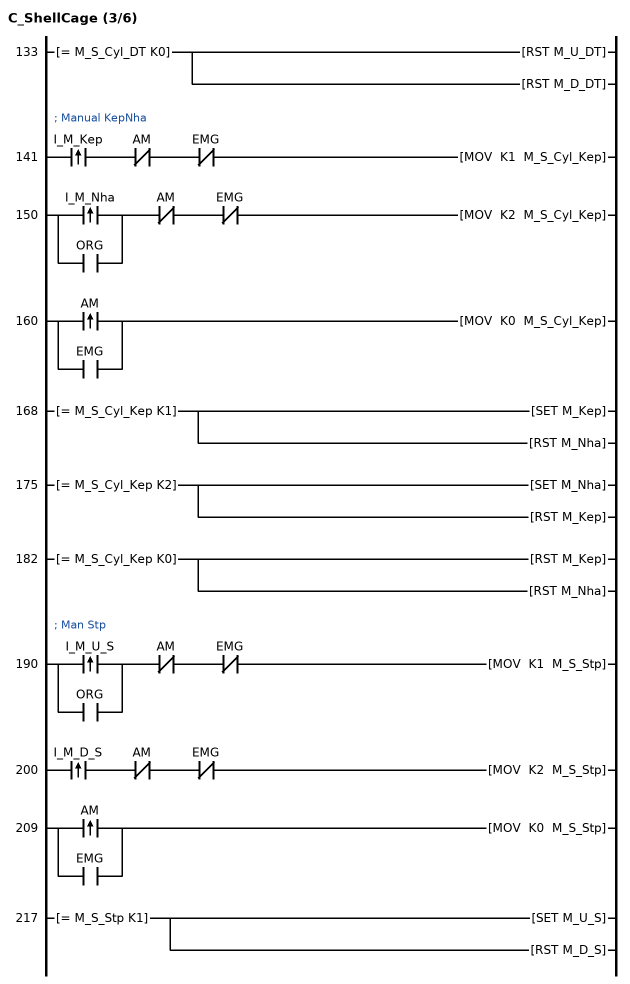
[picture p48: ladder of C_ShellCage, rungs at steps 133 to 217]
133   LD=     M_S_Cyl_DT K0
      RST     M_U_DT
      RST     M_D_DT
; Manual KepNha
141   LDP     I_M_Kep
      ANI     AM
      ANI     EMG
      MOV     K1 M_S_Cyl_Kep
150   LDP     I_M_Nha
      OR      ORG
      ANI     AM
      ANI     EMG
      MOV     K2 M_S_Cyl_Kep
160   LDP     AM
      OR      EMG
      MOV     K0 M_S_Cyl_Kep
168   LD=     M_S_Cyl_Kep K1
      SET     M_Kep
      RST     M_Nha
175   LD=     M_S_Cyl_Kep K2
      SET     M_Nha
      RST     M_Kep
182   LD=     M_S_Cyl_Kep K0
      RST     M_Kep
      RST     M_Nha
; Man Stp
190   LDP     I_M_U_S
      OR      ORG
      ANI     AM
      ANI     EMG
      MOV     K1 M_S_Stp
200   LDP     I_M_D_S
      ANI     AM
      ANI     EMG
      MOV     K2 M_S_Stp
209   LDP     AM
      OR      EMG
      MOV     K0 M_S_Stp
217   LD=     M_S_Stp K1
      SET     M_U_S
      RST     M_D_S
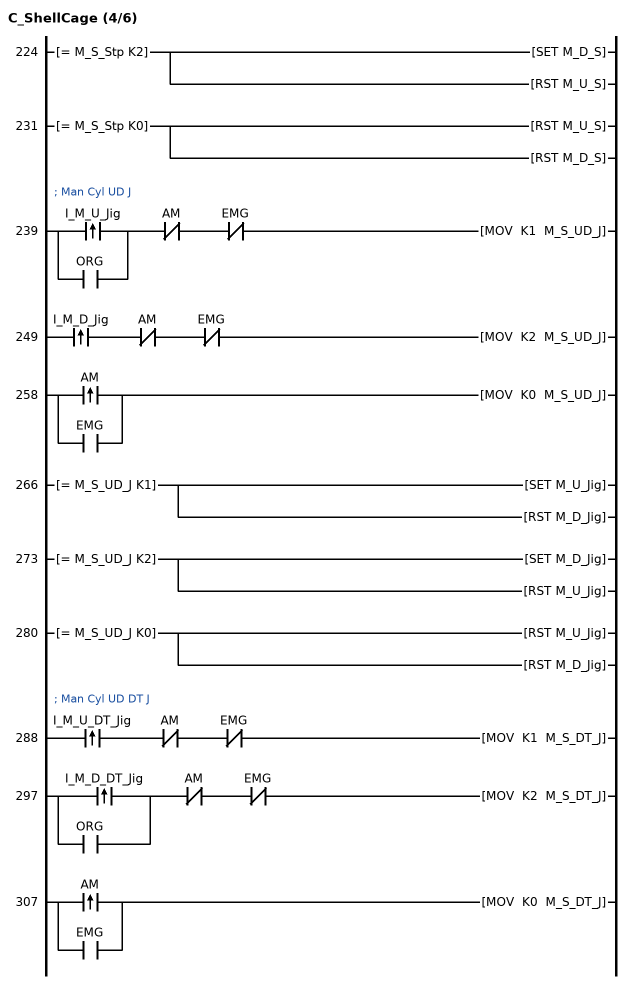
224   LD=     M_S_Stp K2
      SET     M_D_S
      RST     M_U_S
231   LD=     M_S_Stp K0
      RST     M_U_S
      RST     M_D_S
; Man Cyl UD J
239   LDP     I_M_U_Jig
      OR      ORG
      ANI     AM
      ANI     EMG
      MOV     K1 M_S_UD_J
249   LDP     I_M_D_Jig
      ANI     AM
      ANI     EMG
      MOV     K2 M_S_UD_J
258   LDP     AM
      OR      EMG
      MOV     K0 M_S_UD_J
266   LD=     M_S_UD_J K1
      SET     M_U_Jig
      RST     M_D_Jig
273   LD=     M_S_UD_J K2
      SET     M_D_Jig
      RST     M_U_Jig
280   LD=     M_S_UD_J K0
      RST     M_U_Jig
      RST     M_D_Jig
; Man Cyl UD DT J
288   LDP     I_M_U_DT_Jig
      ANI     AM
      ANI     EMG
      MOV     K1 M_S_DT_J
297   LDP     I_M_D_DT_Jig
      OR      ORG
      ANI     AM
      ANI     EMG
      MOV     K2 M_S_DT_J
307   LDP     AM
      OR      EMG
      MOV     K0 M_S_DT_J
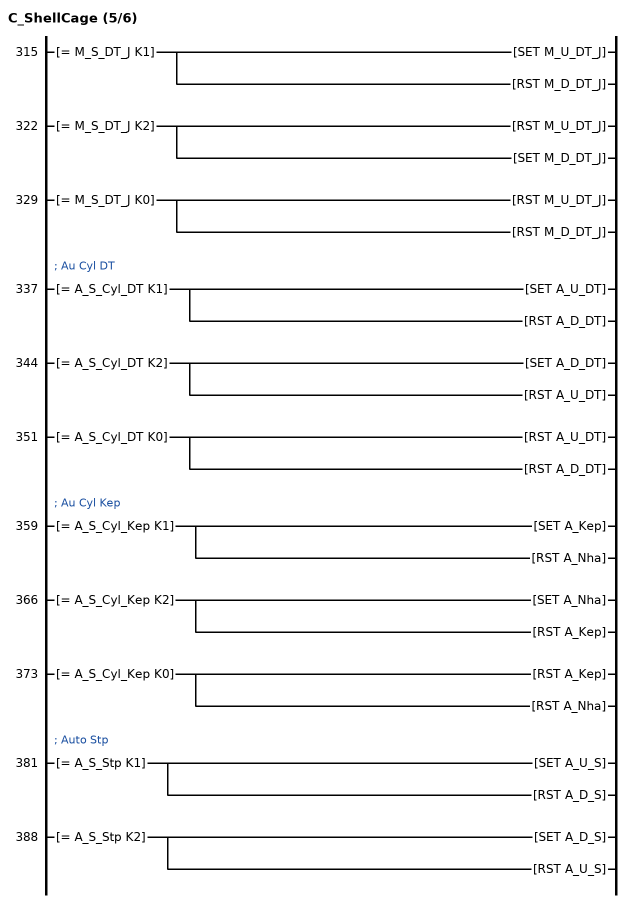
315   LD=     M_S_DT_J K1
      SET     M_U_DT_J
      RST     M_D_DT_J
322   LD=     M_S_DT_J K2
      RST     M_U_DT_J
      SET     M_D_DT_J
329   LD=     M_S_DT_J K0
      RST     M_U_DT_J
      RST     M_D_DT_J
; Au Cyl DT
337   LD=     A_S_Cyl_DT K1
      SET     A_U_DT
      RST     A_D_DT
344   LD=     A_S_Cyl_DT K2
      SET     A_D_DT
      RST     A_U_DT
351   LD=     A_S_Cyl_DT K0
      RST     A_U_DT
      RST     A_D_DT
; Au Cyl Kep
359   LD=     A_S_Cyl_Kep K1
      SET     A_Kep
      RST     A_Nha
366   LD=     A_S_Cyl_Kep K2
      SET     A_Nha
      RST     A_Kep
373   LD=     A_S_Cyl_Kep K0
      RST     A_Kep
      RST     A_Nha
; Auto Stp
381   LD=     A_S_Stp K1
      SET     A_U_S
      RST     A_D_S
388   LD=     A_S_Stp K2
      SET     A_D_S
      RST     A_U_S
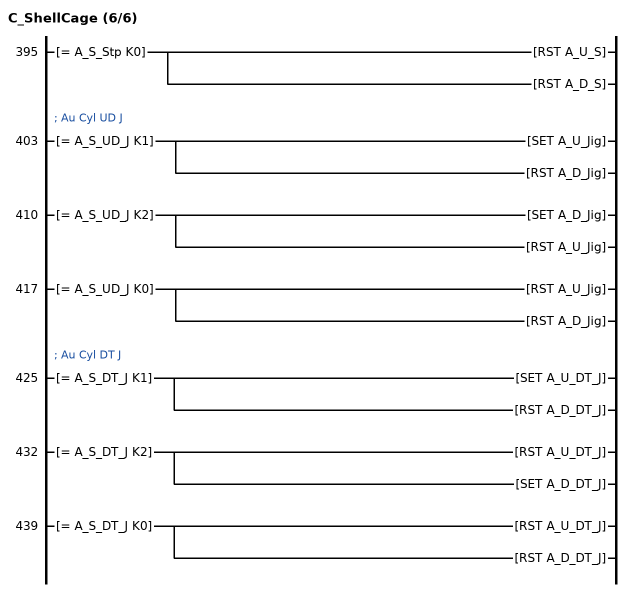
395   LD=     A_S_Stp K0
      RST     A_U_S
      RST     A_D_S
; Au Cyl UD J
403   LD=     A_S_UD_J K1
      SET     A_U_Jig
      RST     A_D_Jig
410   LD=     A_S_UD_J K2
      SET     A_D_Jig
      RST     A_U_Jig
417   LD=     A_S_UD_J K0
      RST     A_U_Jig
      RST     A_D_Jig
; Au Cyl DT J
425   LD=     A_S_DT_J K1
      SET     A_U_DT_J
      RST     A_D_DT_J
432   LD=     A_S_DT_J K2
      RST     A_U_DT_J
      SET     A_D_DT_J
439   LD=     A_S_DT_J K0
      RST     A_U_DT_J
      RST     A_D_DT_J
END_FUNCTION_BLOCK

PROGRAM Position
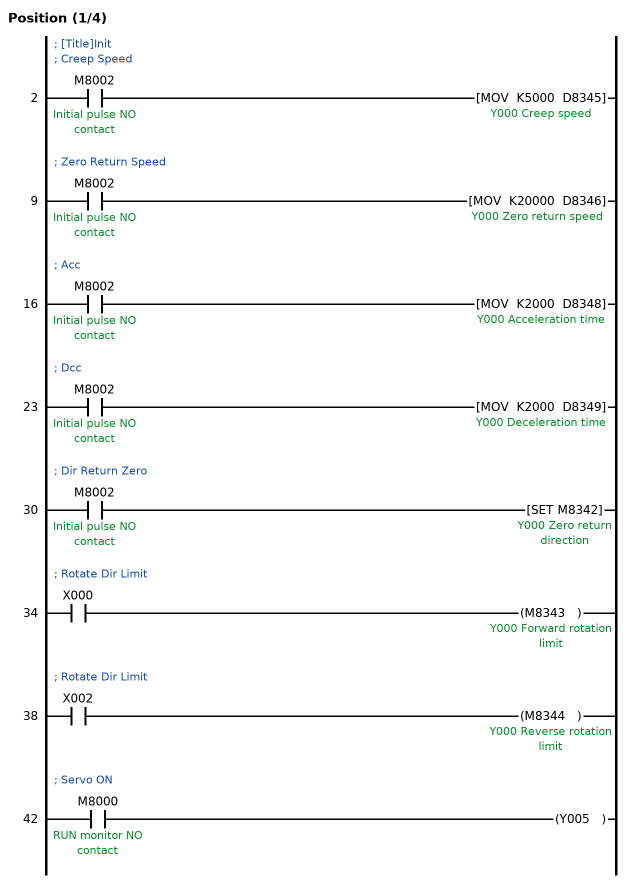
; [Title]Init
; Creep Speed
2     LD      M8002  ; Initial pulse NO contact
      MOV     K5000 D8345  ; Y000 Creep speed
; Zero Return Speed
9     LD      M8002  ; Initial pulse NO contact
      MOV     K20000 D8346  ; Y000 Zero return speed
; Acc
16    LD      M8002  ; Initial pulse NO contact
      MOV     K2000 D8348  ; Y000 Acceleration time
; Dcc
23    LD      M8002  ; Initial pulse NO contact
      MOV     K2000 D8349  ; Y000 Deceleration time
; Dir Return Zero
30    LD      M8002  ; Initial pulse NO contact
      SET     M8342  ; Y000 Zero return direction
; Rotate Dir Limit
34    LD      X000
      OUT     M8343  ; Y000 Forward rotation limit
; Rotate Dir Limit
38    LD      X002
      OUT     M8344  ; Y000 Reverse rotation limit
; Servo ON
42    LD      M8000  ; RUN monitor NO contact
      OUT     Y005
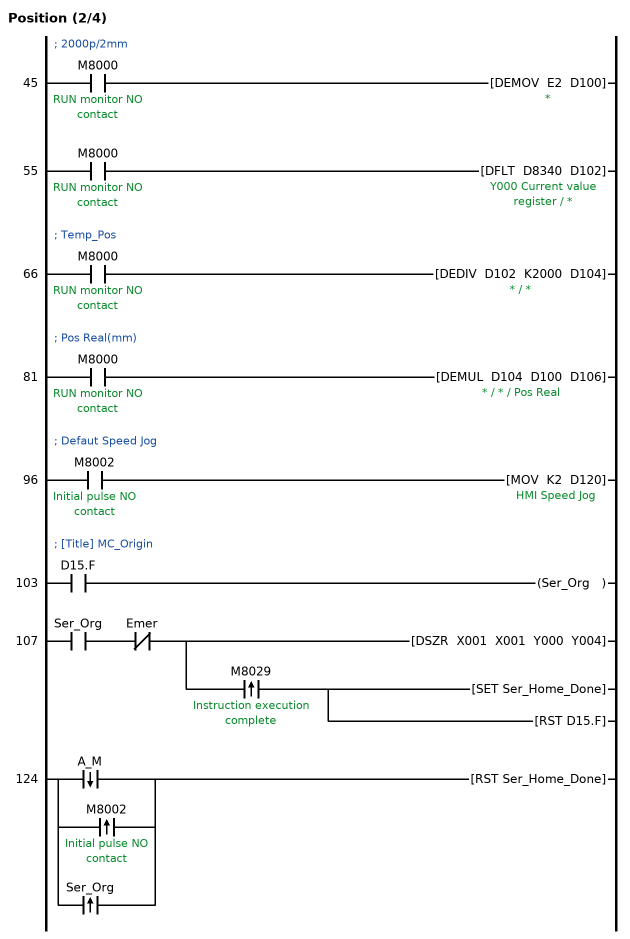
; 2000p/2mm
45    LD      M8000  ; RUN monitor NO contact
      DEMOV   E2 D100  ; *
55    LD      M8000  ; RUN monitor NO contact
      DFLT    D8340 D102  ; Y000 Current value register / *
; Temp_Pos
66    LD      M8000  ; RUN monitor NO contact
      DEDIV   D102 K2000 D104  ; *
; Pos Real(mm)
81    LD      M8000  ; RUN monitor NO contact
      DEMUL   D104 D100 D106  ; Pos Real
; Defaut Speed Jog
96    LD      M8002  ; Initial pulse NO contact
      MOV     K2 D120  ; HMI Speed Jog
; [Title] MC_Origin
103   LD      D15.F
      OUT     Ser_Org
107   LD      Ser_Org
      ANI     Emer
      DSZR    X001 X001 Y000 Y004
      ANDP    M8029  ; Instruction execution complete
      SET     Ser_Home_Done
      RST     D15.F
124   LDF     A_M
      ORP     M8002  ; Initial pulse NO contact
      ORP     Ser_Org
      RST     Ser_Home_Done
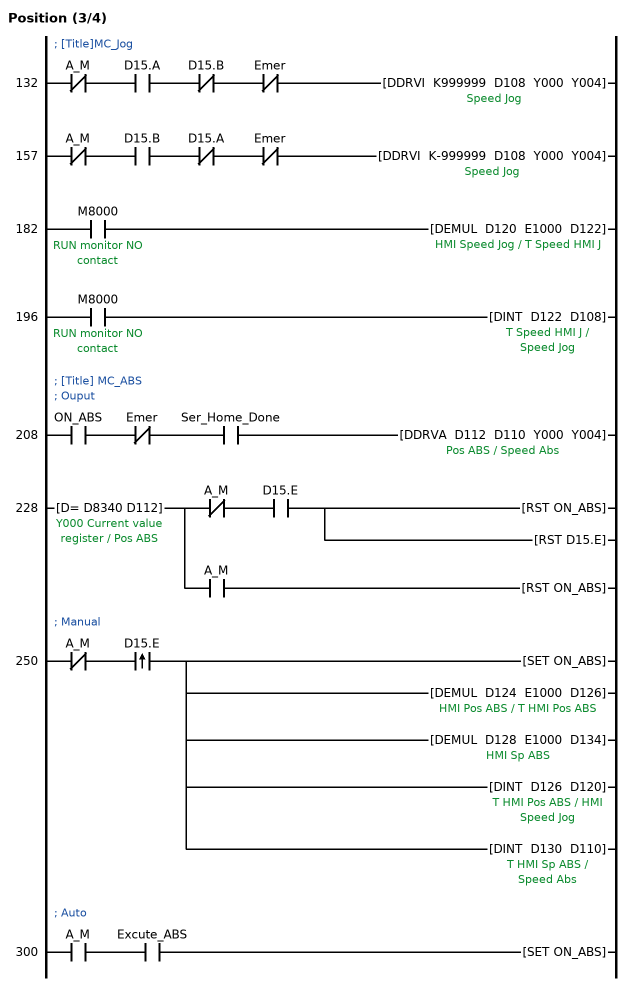
; [Title]MC_Jog
132   LDI     A_M
      AND     D15.A
      ANI     D15.B
      ANI     Emer
      DDRVI   K999999 D108 Y000 Y004  ; Speed Jog
157   LDI     A_M
      AND     D15.B
      ANI     D15.A
      ANI     Emer
      DDRVI   K-999999 D108 Y000 Y004
182   LD      M8000  ; RUN monitor NO contact
      DEMUL   D120 E1000 D122  ; T Speed HMI J
196   LD      M8000  ; RUN monitor NO contact
      DINT    D122 D108
; [Title] MC_ABS
; Ouput
208   LD      ON_ABS
      ANI     Emer
      AND     Ser_Home_Done
      DDRVA   D112 D110 Y000 Y004  ; Pos ABS / Speed Abs
228   LDD=    D8340 D112  ; Y000 Current value register / Pos ABS
      MPS
      ANI     A_M
      AND     D15.E
      RST     ON_ABS
      RST     D15.E
      MPP
      AND     A_M
      RST     ON_ABS
; Manual
250   LDI     A_M
      ANDP    D15.E
      SET     ON_ABS
      DEMUL   D124 E1000 D126  ; HMI Pos ABS / T HMI Pos ABS
      DEMUL   D128 E1000 D134  ; HMI Sp ABS
      DINT    D126 D120
      DINT    D130 D110  ; T HMI Sp ABS
; Auto
300   LD      A_M
      AND     Excute_ABS
      SET     ON_ABS
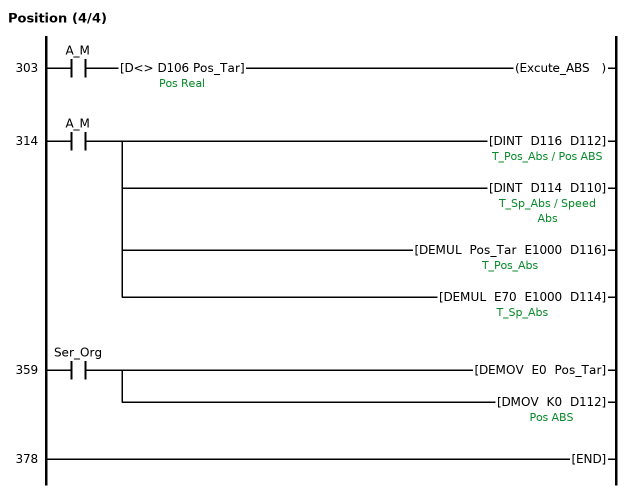
303   LD      A_M
      ANDD<>  D106 Pos_Tar  ; Pos Real
      OUT     Excute_ABS
314   LD      A_M
      DINT    D116 D112  ; T_Pos_Abs
      DINT    D114 D110  ; T_Sp_Abs
      DEMUL   Pos_Tar E1000 D116
      DEMUL   E70 E1000 D114
359   LD      Ser_Org
      DEMOV   E0 Pos_Tar
      DMOV    K0 D112
378   END
END_PROGRAM

PROGRAM Input
VAR
  D_M47 : TIMER;
END_VAR
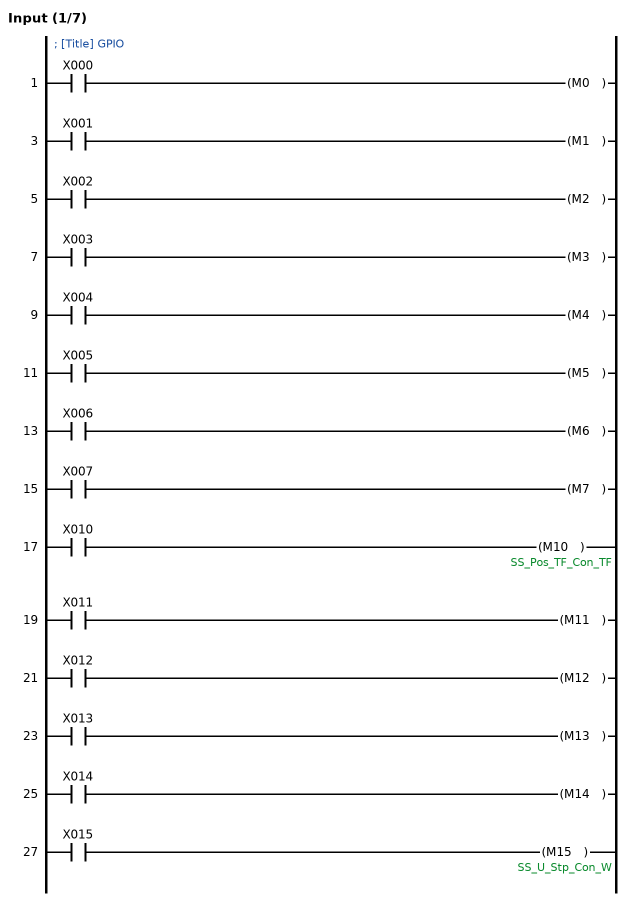
; [Title] GPIO
1     LD      X000
      OUT     M0
3     LD      X001
      OUT     M1
5     LD      X002
      OUT     M2
7     LD      X003
      OUT     M3
9     LD      X004
      OUT     M4
11    LD      X005
      OUT     M5
13    LD      X006
      OUT     M6
15    LD      X007
      OUT     M7
17    LD      X010
      OUT     M10  ; SS_Pos_TF_Con_TF
19    LD      X011
      OUT     M11
21    LD      X012
      OUT     M12
23    LD      X013
      OUT     M13
25    LD      X014
      OUT     M14
27    LD      X015
      OUT     M15  ; SS_U_Stp_Con_W
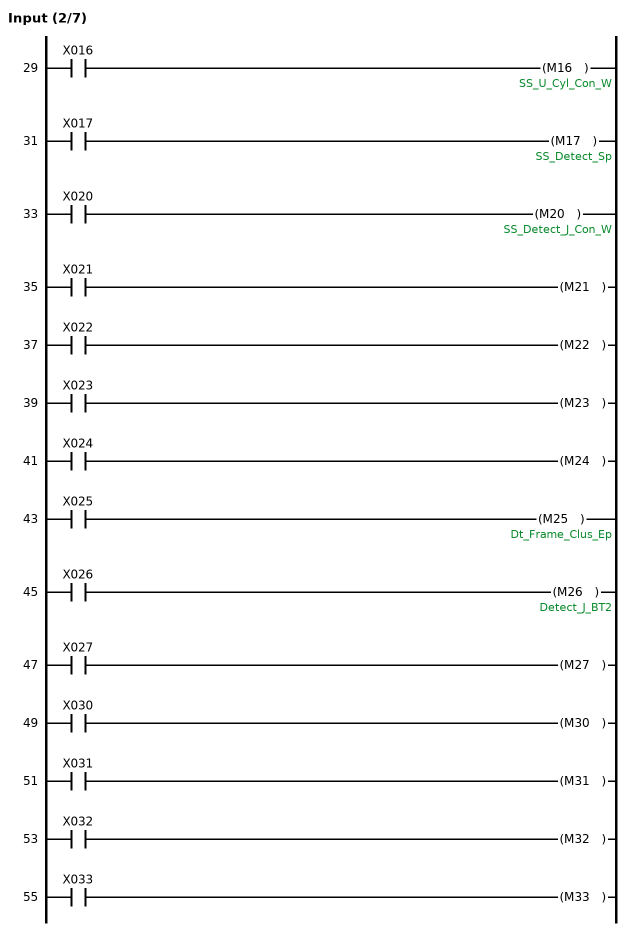
29    LD      X016
      OUT     M16  ; SS_U_Cyl_Con_W
31    LD      X017
      OUT     M17  ; SS_Detect_Sp
33    LD      X020
      OUT     M20  ; SS_Detect_J_Con_W
35    LD      X021
      OUT     M21
37    LD      X022
      OUT     M22
39    LD      X023
      OUT     M23
41    LD      X024
      OUT     M24
43    LD      X025
      OUT     M25  ; Dt_Frame_Clus_Ep
45    LD      X026
      OUT     M26  ; Detect_J_BT2
47    LD      X027
      OUT     M27
49    LD      X030
      OUT     M30
51    LD      X031
      OUT     M31
53    LD      X032
      OUT     M32
55    LD      X033
      OUT     M33
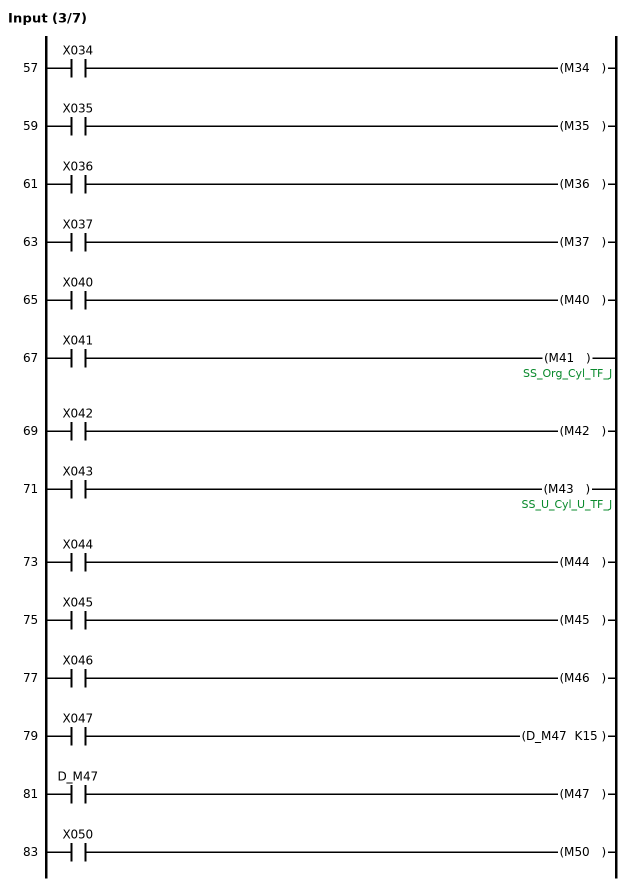
57    LD      X034
      OUT     M34
59    LD      X035
      OUT     M35
61    LD      X036
      OUT     M36
63    LD      X037
      OUT     M37
65    LD      X040
      OUT     M40
67    LD      X041
      OUT     M41  ; SS_Org_Cyl_TF_J
69    LD      X042
      OUT     M42
71    LD      X043
      OUT     M43  ; SS_U_Cyl_U_TF_J
73    LD      X044
      OUT     M44
75    LD      X045
      OUT     M45
77    LD      X046
      OUT     M46
79    LD      X047
      OUT     D_M47 K15
81    LD      D_M47
      OUT     M47
83    LD      X050
      OUT     M50
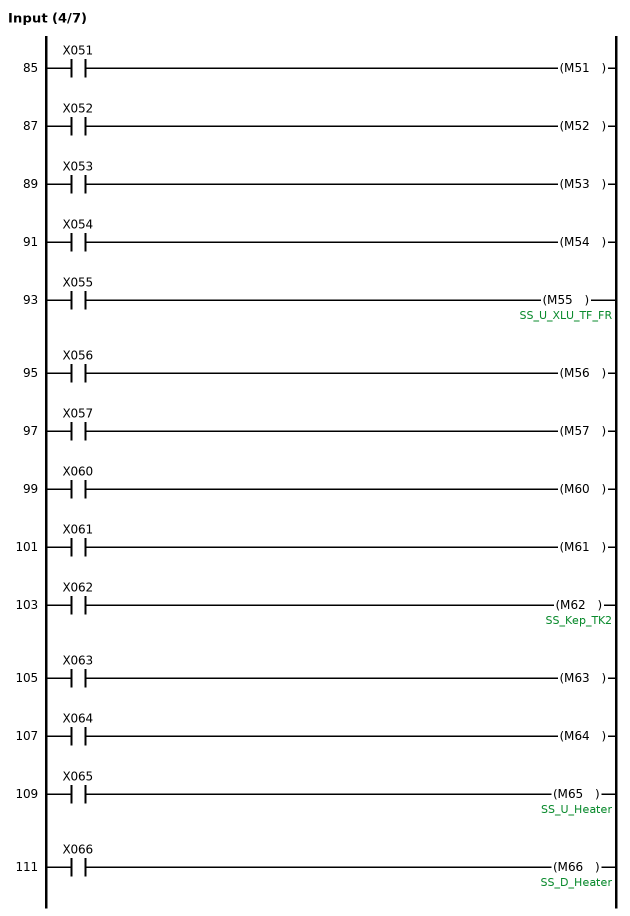
85    LD      X051
      OUT     M51
87    LD      X052
      OUT     M52
89    LD      X053
      OUT     M53
91    LD      X054
      OUT     M54
93    LD      X055
      OUT     M55  ; SS_U_XLU_TF_FR
95    LD      X056
      OUT     M56
97    LD      X057
      OUT     M57
99    LD      X060
      OUT     M60
101   LD      X061
      OUT     M61
103   LD      X062
      OUT     M62  ; SS_Kep_TK2
105   LD      X063
      OUT     M63
107   LD      X064
      OUT     M64
109   LD      X065
      OUT     M65  ; SS_U_Heater
111   LD      X066
      OUT     M66  ; SS_D_Heater
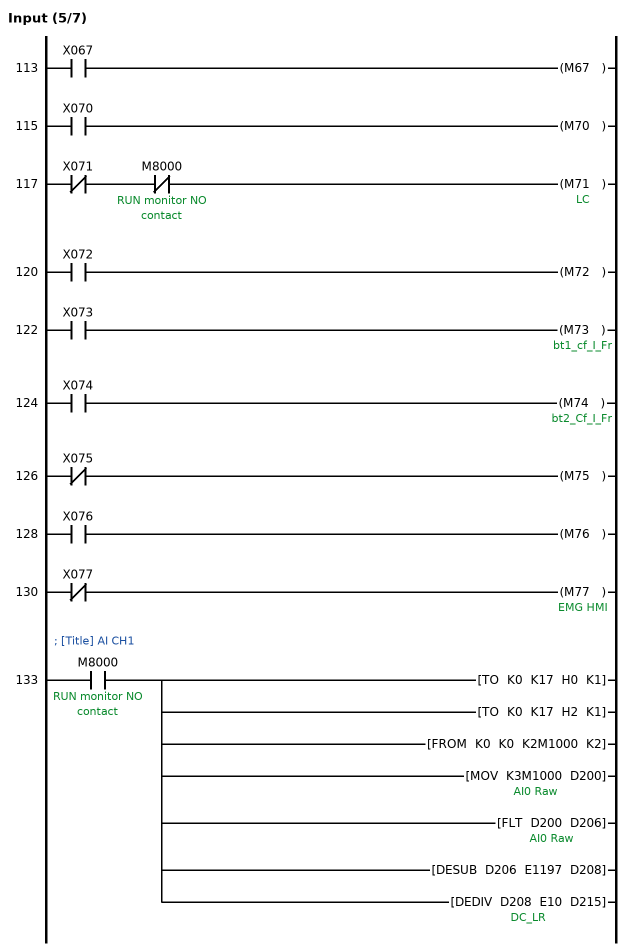
113   LD      X067
      OUT     M67
115   LD      X070
      OUT     M70
117   LDI     X071
      ANI     M8000  ; RUN monitor NO contact
      OUT     M71  ; LC
120   LD      X072
      OUT     M72
122   LD      X073
      OUT     M73  ; bt1_cf_I_Fr
124   LD      X074
      OUT     M74  ; bt2_Cf_I_Fr
126   LDI     X075
      OUT     M75
128   LD      X076
      OUT     M76
130   LDI     X077
      OUT     M77  ; EMG HMI
; [Title] AI CH1
133   LD      M8000  ; RUN monitor NO contact
      TO      K0 K17 H0 K1
      TO      K0 K17 H2 K1
      FROM    K0 K0 K2M1000 K2
      MOV     K3M1000 D200  ; AI0 Raw
      FLT     D200 D206
      DESUB   D206 E1197 D208
      DEDIV   D208 E10 D215  ; DC_LR
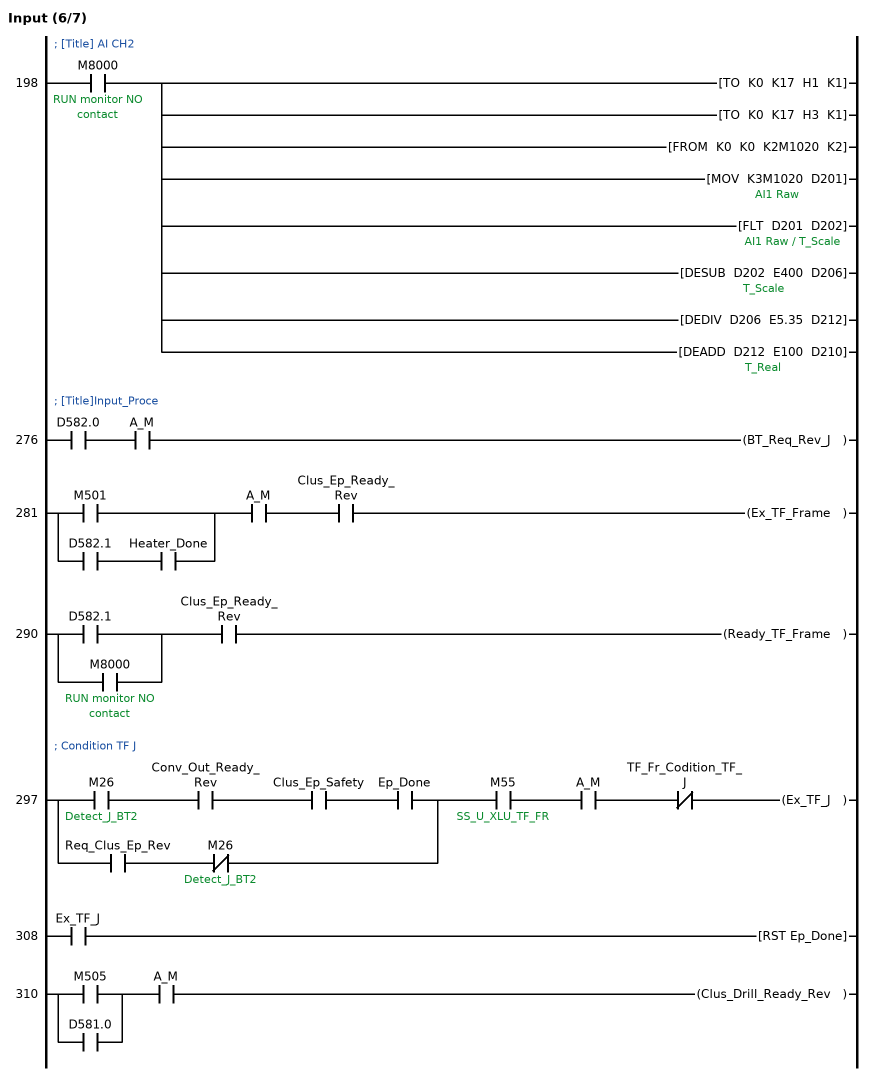
; [Title] AI CH2
198   LD      M8000  ; RUN monitor NO contact
      TO      K0 K17 H1 K1
      TO      K0 K17 H3 K1
      FROM    K0 K0 K2M1020 K2
      MOV     K3M1020 D201  ; AI1 Raw
      FLT     D201 D202  ; T_Scale
      DESUB   D202 E400 D206
      DEDIV   D206 E5.35 D212
      DEADD   D212 E100 D210  ; T_Real
; [Title]Input_Proce
276   LD      D582.0
      AND     A_M
      OUT     BT_Req_Rev_J
281   LD      M501
      LD      D582.1
      AND     Heater_Done
      ORB
      AND     A_M
      AND     Clus_Ep_Ready_Rev
      OUT     Ex_TF_Frame
290   LD      D582.1
      OR      M8000  ; RUN monitor NO contact
      AND     Clus_Ep_Ready_Rev
      OUT     Ready_TF_Frame
; Condition TF J
297   LD      M26  ; Detect_J_BT2
      AND     Conv_Out_Ready_Rev
      AND     Clus_Ep_Safety
      AND     Ep_Done
      LD      Req_Clus_Ep_Rev
      ANI     M26  ; Detect_J_BT2
      ORB
      AND     M55  ; SS_U_XLU_TF_FR
      AND     A_M
      ANI     TF_Fr_Codition_TF_J
      OUT     Ex_TF_J
308   LD      Ex_TF_J
      RST     Ep_Done
310   LD      M505
      OR      D581.0
      AND     A_M
      OUT     Clus_Drill_Ready_Rev
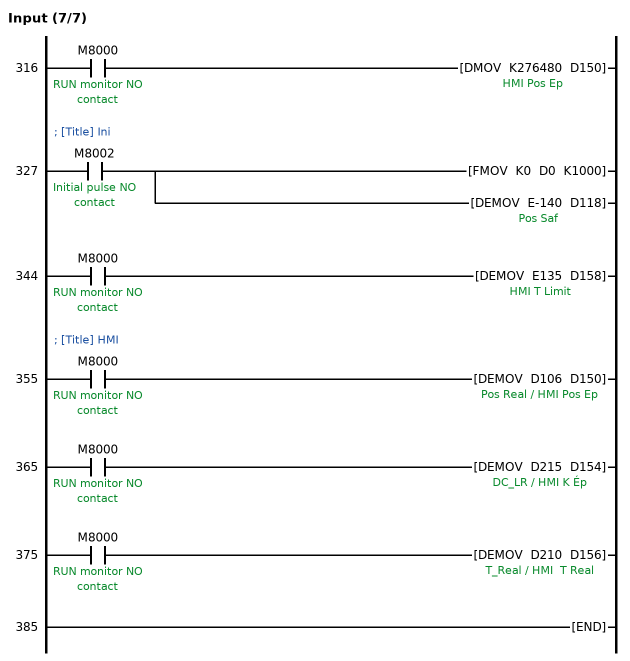
316   LD      M8000  ; RUN monitor NO contact
      DMOV    K276480 D150  ; HMI Pos Ep
; [Title] Ini
327   LD      M8002  ; Initial pulse NO contact
      FMOV    K0 D0 K1000
      DEMOV   E-140 D118  ; Pos Saf
344   LD      M8000  ; RUN monitor NO contact
      DEMOV   E135 D158  ; HMI T Limit
; [Title] HMI
355   LD      M8000  ; RUN monitor NO contact
      DEMOV   D106 D150  ; Pos Real
365   LD      M8000  ; RUN monitor NO contact
      DEMOV   D215 D154  ; HMI K Ép
375   LD      M8000  ; RUN monitor NO contact
      DEMOV   D210 D156  ; HMI  T Real
385   END
END_PROGRAM

PROGRAM EMG
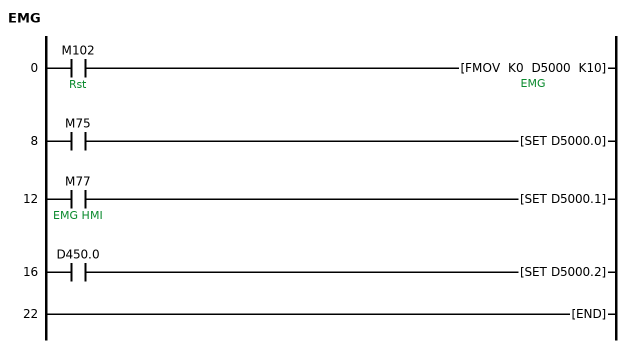
0     LD      M102  ; Rst
      FMOV    K0 D5000 K10  ; EMG
8     LD      M75
      SET     D5000.0
12    LD      M77  ; EMG HMI
      SET     D5000.1
16    LD      D450.0
      SET     D5000.2
22    END
END_PROGRAM

PROGRAM Order
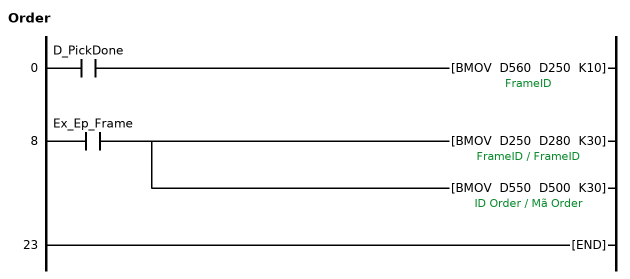
0     LD      D_PickDone
      BMOV    D560 D250 K10  ; FrameID
8     LD      Ex_Ep_Frame
      BMOV    D250 D280 K30  ; FrameID
      BMOV    D550 D500 K30  ; ID Order / Mã Order
23    END
END_PROGRAM

// device comments not shown above
D152  ; HMI Sp ABS
D160  ; Spare
D249  ; /*Data in
D260  ; DC TC
D264  ; Pos Kep
D266  ; Pos Ep
D279  ; /*Data Out
D292  ; T Target
D499  ; Master
D520  ; Status
D522  ; Value 1
D523  ; Value 2
D532  ; S_Tranfer
D570  ; ID Frame
D590  ; S_Tranfer
D5001  ; ALARM
